% RSLogix 500 project I2P Job 10 - Tyler_Vogt.RSS, saved by version 10.00.00.00 %
PROJECT "MLO2B"    % processor: Bul.1763 MicroLogix 1100 Series B %

PROGRAM FILES
  LAD 2   5 rungs

DATA FILES
  O0 OUTPUT  4 elements
  I1 INPUT  6 elements
  S2 STATUS  66 elements
  B3 BINARY  1 elements
  T4 TIMER  1 elements
  C5 COUNTER  1 elements
  R6 CONTROL  1 elements
  N7 INTEGER  1 elements
  F8 FLOAT  1 elements

LADDER 2
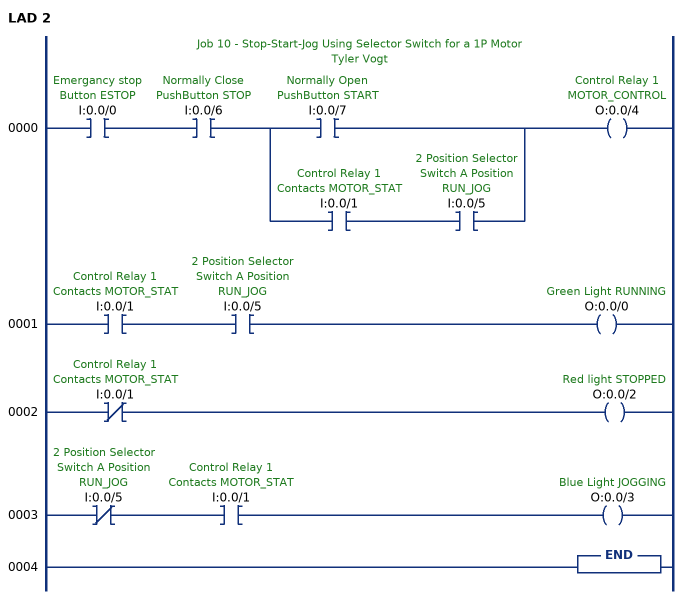
% Rung: 0 %
% Job 10 - Stop-Start-Jog Using Selector Switch for a 1P Motor
% Tyler Vogt %
SOR XIC I:0.0/0 XIC I:0.0/6 BST XIC I:0.0/7 NXB XIC I:0.0/1 XIC I:0.0/5 BND OTE O:0.0/4 EOR
%   I:0.0/0  ESTOP  "Emergancy stop Button" %
%   I:0.0/6  STOP  "Normally Close PushButton" %
%   I:0.0/7  START  "Normally Open PushButton" %
%   I:0.0/1  MOTOR_STAT  "Control Relay 1 Contacts" %
%   I:0.0/5  RUN_JOG  "2 Position Selector Switch A Position" %
%   O:0.0/4  MOTOR_CONTROL  "Control Relay 1" %
% Rung: 1 %
SOR XIC I:0.0/1 XIC I:0.0/5 OTE O:0.0/0 EOR
%   I:0.0/1  MOTOR_STAT  "Control Relay 1 Contacts" %
%   I:0.0/5  RUN_JOG  "2 Position Selector Switch A Position" %
%   O:0.0/0  RUNNING  "Green Light" %
% Rung: 2 %
SOR XIO I:0.0/1 OTE O:0.0/2 EOR
%   I:0.0/1  MOTOR_STAT  "Control Relay 1 Contacts" %
%   O:0.0/2  STOPPED  "Red light" %
% Rung: 3 %
SOR XIO I:0.0/5 XIC I:0.0/1 OTE O:0.0/3 EOR
%   I:0.0/5  RUN_JOG  "2 Position Selector Switch A Position" %
%   I:0.0/1  MOTOR_STAT  "Control Relay 1 Contacts" %
%   O:0.0/3  JOGGING  "Blue Light" %
% Rung: 4 %
SOR END EOR

OTHER DOCUMENTED ADDRESSES
  I:0.0/2  CR2_STAT  "Control Relay 2 Contacts"
  I:0.0/3  3PSS_A  "3 Position Selector Switch A Position"
  I:0.0/4  3PSS_B  "3 Position Selector Switch B Position"
  I:0.0/8  PB3  "Normally Open PushButton"
  O:0.0/1  YLW_LT  "Yellow Light"
  O:0.0/5  CR2  "Control Relay 2"
